Staubli VAL3: onF6Event.pgx

program onF6Event()
begin
  // look if the bButton is enable
  if bButton[5]
    //
    // PAUSE / RESUME
    //
    if !cycleStatus:bPause
      logMsg("[KERNEL] INTERFACE:Pause cycle")
      call OnEvent:pauseCycle()
    else
      logMsg("[KERNEL] INTERFACE:Resume cycle")
      call OnEvent:resumeCycle()
    endIf
  endIf
end
